Omron CX-Programmer project NewProject (CX-Programmer 9.75)

# PLC NewPLC1: CP1L M

## Global symbols (name address type ; comment)
0.00 BOOL  ; +
0.01 BOOL  ; -
0.02 BOOL  ; *
0.03 BOOL  ; /
0.04 BOOL  ; =
0.05 BOOL  ; Reset
2.00 BOOL  ; Display Buffer
2.01 BOOL  ; Reset
W0.00 BOOL  ; + Operation
W0.01 BOOL  ; - Operation
W0.02 BOOL  ; * Operation
W0.03 BOOL  ; / Operation

## Program NewProgram1 (cyclic task 0)

### Section Section1

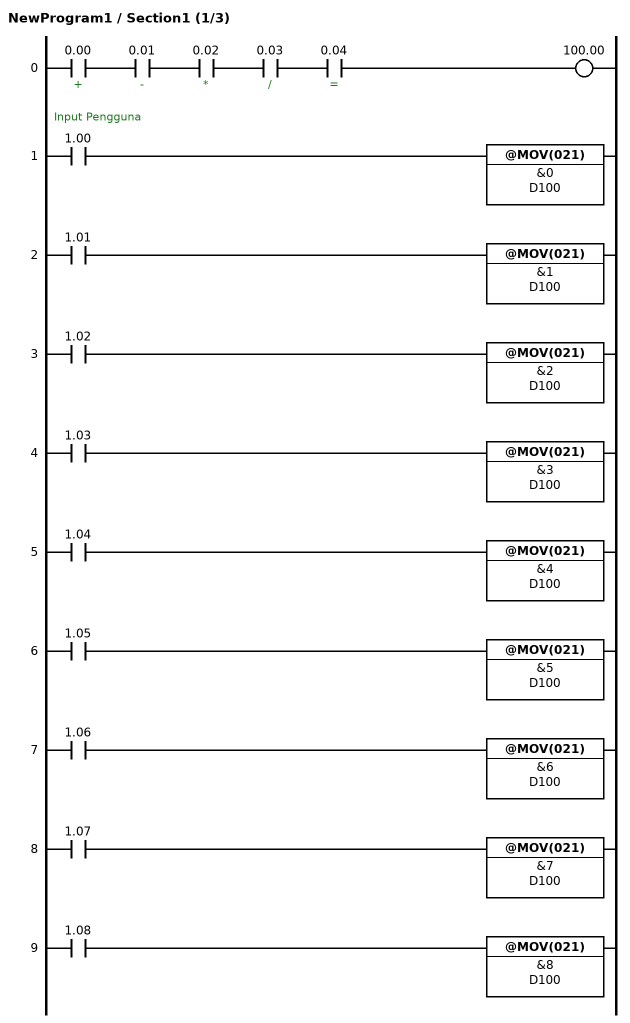
; rung 0
LD 0.00  ; +
AND 0.01  ; -
AND 0.02  ; *
AND 0.03  ; /
AND 0.04  ; =
OUT 100.00
; rung 1: Input Pengguna
LD 1.00
@MOV(021) &0 D100
; rung 2
LD 1.01
@MOV(021) &1 D100
; rung 3
LD 1.02
@MOV(021) &2 D100
; rung 4
LD 1.03
@MOV(021) &3 D100
; rung 5
LD 1.04
@MOV(021) &4 D100
; rung 6
LD 1.05
@MOV(021) &5 D100
; rung 7
LD 1.06
@MOV(021) &6 D100
; rung 8
LD 1.07
@MOV(021) &7 D100
; rung 9
LD 1.08
@MOV(021) &8 D100

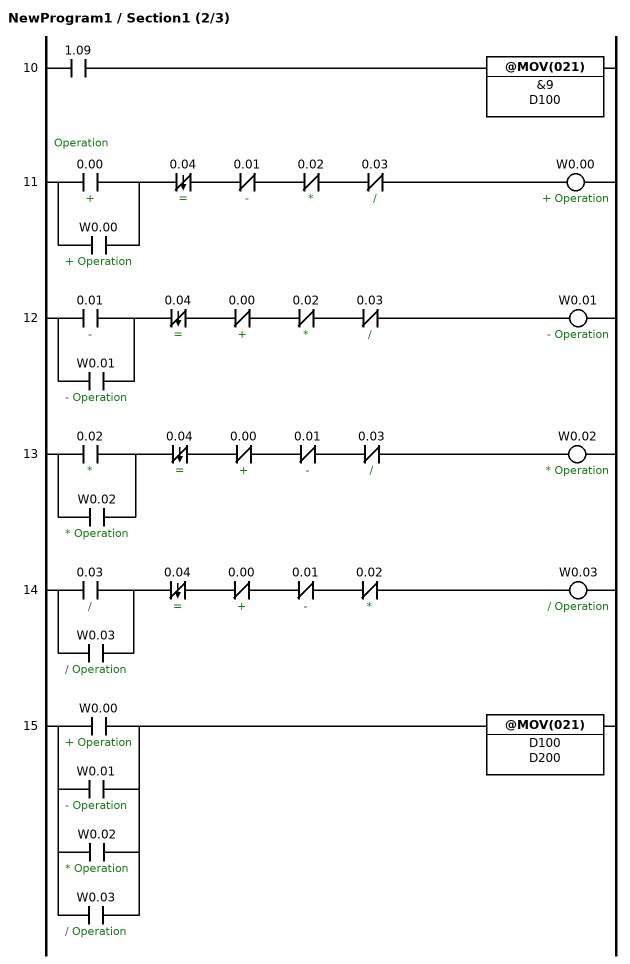
; rung 10
LD 1.09
@MOV(021) &9 D100
; rung 11: Operation
LD 0.00  ; +
OR W0.00  ; + Operation
%ANDNOT 0.04  ; =
ANDNOT 0.01  ; -
ANDNOT 0.02  ; *
ANDNOT 0.03  ; /
OUT W0.00  ; + Operation
; rung 12
LD 0.01  ; -
OR W0.01  ; - Operation
%ANDNOT 0.04  ; =
ANDNOT 0.00  ; +
ANDNOT 0.02  ; *
ANDNOT 0.03  ; /
OUT W0.01  ; - Operation
; rung 13
LD 0.02  ; *
OR W0.02  ; * Operation
%ANDNOT 0.04  ; =
ANDNOT 0.00  ; +
ANDNOT 0.01  ; -
ANDNOT 0.03  ; /
OUT W0.02  ; * Operation
; rung 14
LD 0.03  ; /
OR W0.03  ; / Operation
%ANDNOT 0.04  ; =
ANDNOT 0.00  ; +
ANDNOT 0.01  ; -
ANDNOT 0.02  ; *
OUT W0.03  ; / Operation
; rung 15
LD W0.00  ; + Operation
OR W0.01  ; - Operation
OR W0.02  ; * Operation
OR W0.03  ; / Operation
@MOV(021) D100 D200

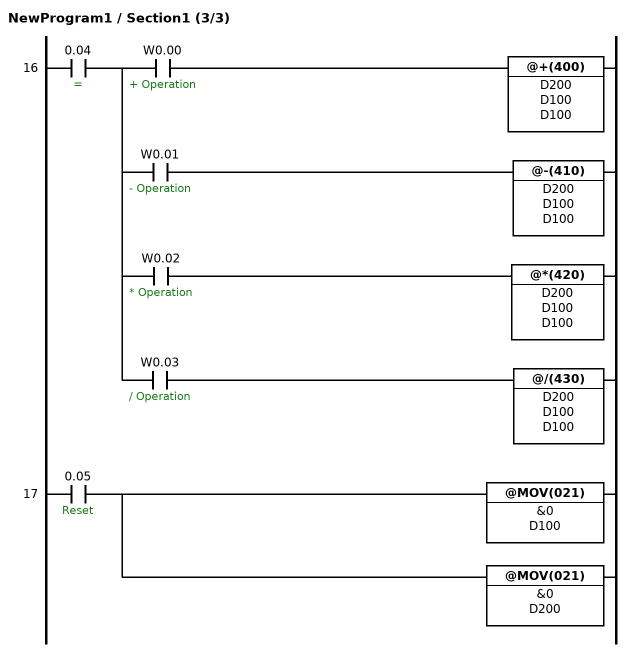
; rung 16
LD 0.04  ; =
OUT TR0
AND W0.00  ; + Operation
@+(400) D200 D100 D100
LD TR0
AND W0.01  ; - Operation
@-(410) D200 D100 D100
LD TR0
AND W0.02  ; * Operation
@*(420) D200 D100 D100
LD TR0
AND W0.03  ; / Operation
@/(430) D200 D100 D100
; rung 17
LD 0.05  ; Reset
@MOV(021) &0 D100
@MOV(021) &0 D200

### Section END
; rung 0
END(001)